FUNCTION_BLOCK FB_LamparaComputada_LD
VAR_INPUT
    ManiobrasTotales: UINT := 2;
END_VAR
VAR_OUTPUT
    ManiobrasPendientes: UINT;
END_VAR
VAR
    Contador: CTD := (CV := ManiobrasTotales);

    Lampara AT %Q*: BOOL;
    Pulsador AT %I*: BOOL;
    PulsadorReinicio AT %I*: BOOL;
END_VAR

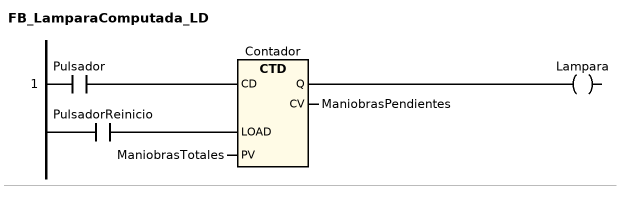
// NETWORK 1
Contador(CD := Pulsador, LOAD := PulsadorReinicio, PV := ManiobrasTotales, CV => ManiobrasPendientes); // CTD
Lampara := Contador.Q;

END_FUNCTION_BLOCK

(* stored: Version 1.1.0.1, ProductVersion 3.1.4024.15
   POU FB_LamparaComputada_LD: Id {41ef2a50-6ccd-433b-b47c-8214546b0362}, SpecialFunc None *)
